FUNCTION_BLOCK HnhtHnltLinkage
VAR_INPUT
END_VAR
VAR_OUTPUT
END_VAR
VAR
END_VAR

END_FUNCTION_BLOCK

(* stored: Version 1.1.0.1, ProductVersion 3.1.4024.10
   POU HnhtHnltLinkage: Id {6a3baad8-61ea-416c-a36f-d39a6e6cabde}, SpecialFunc None *)
